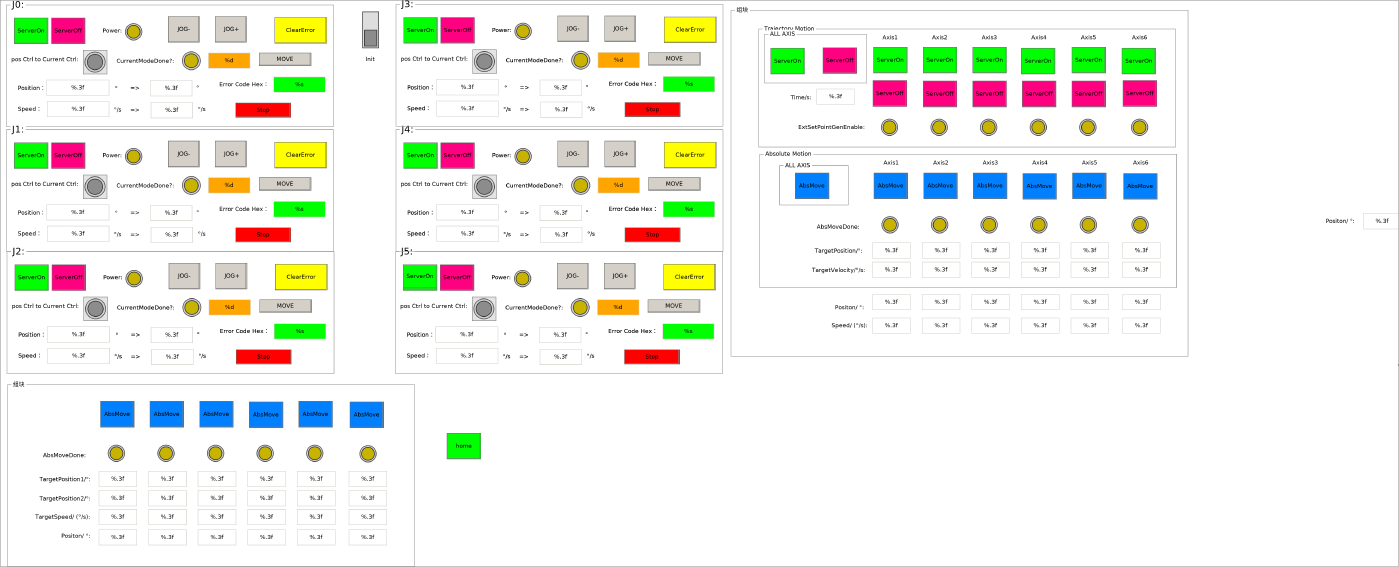
VISUALIZATION StatJoint_6Axis  // 2680x1087
    GroupBox (12,1 627x242), "J0:"
        Label (6,94 136x38), "pos Ctrl to Current Ctrl:"
        Label (13,192 64x32), "Speed："
        Label (224,191 45x38), "=>"
        Textfield (77,152 120x30), "%.3f", text variable: MAIN.AxisInfo[0].PositionCmd
        Label (198,154 22x29), "°"
        Textfield (78,193 119x30), "%.3f", text variable: MAIN.AxisMotionPara[0].TargetVelocity
            OnMouseClick: write the text variable via VisuDialogs.Numpad
        Label (193,195 37x29), "°/s"
        Button (86,33 65x50), "ServerOff", input disabled if: NOT MAIN.AxisOp[0].AxisInfo.AxisStatus.Ready
            toggle MAIN.HMI_AxisEnable[0]
        Button (514,32 100x50), "ClearError"
            tap MAIN.HMI_Axis_reset[0]
        Label (173,43 60x30), "Power:"
        Label (261,47 40x30)
        Button (310,30 60x50), "JOG-"
            tap MAIN.HMI_AxisJogBackwards[0]
        Button (400,30 60x50), "JOG+"
            tap MAIN.HMI_AxisJogFoward[0]
        Textfield (276,153 80x30), "%.3f", text variable: MAIN.AxisInfo[0].ActualPosition
        Label (354,153 22x29), "°"
        Label (354,194 37x29), "°/s"
        Textfield (277,195 80x30), "%.3f", text variable: MAIN.AxisInfo[0].ActualVelocity
        Textfield (387,100 80x30), "%d", text variable: MAIN.HMI_TargetTorque[0]
            OnMouseClick: write the text variable via VisuDialogs.Numpad
        Button (484,100 100x25), "MOVE"
            toggle MAIN.HMI_CurrentControlMove[0]
        Label (406,146 99x30), "Error Code Hex："
        Textfield (512,146 99x30), "%s", text variable: MAIN.AxisOp[0].AxisInfo.ErrId_Hex
        Label (224,149 45x38), "=>"
        Button (15,33 65x50), "ServerOn", input disabled if: NOT MAIN.AxisOp[0].AxisInfo.AxisStatus.Ready
            toggle MAIN.HMI_AxisEnable[0]
        PushSwitchLed (146,95 48x46), variable: MAIN.HMI_CurrentControlOfEnable[0], behaviour: TOGGLE, style: Switch-PushSwitchLed-Gray
        Label (18,149 62x38), "Position："
        Button (439,196 106x28), "Stop"
            tap MAIN.HMI_AxisStop[0]
        Lamp1 (225,40 38x40), variable: MAIN.AxisOp[0].AxisInfo.AxisStatus.Enabled, style: Lamp-Lamp1-Yellow
        Label (209,97 115x38), "CurrentModeDone?:"
        Lamp1 (334,94 41x43), variable: MAIN.HMI_AxisCurrentControlFlag[0], style: Lamp-Lamp1-Yellow
        Textfield (78,625 120x30), "%.3f", text variable: MAIN.AxisInfo[0].PositionCmd
        Label (199,627 22x29), "°"
        Label (14,665 64x32), "Speed："
        Textfield (79,666 119x30), "%.3f", text variable: MAIN.AxisMotionPara[0].TargetVelocity
            OnMouseClick: write the text variable via VisuDialogs.Numpad
        Label (194,668 37x29), "°/s"
        Button (87,506 65x50), "ServerOff", input disabled if: NOT MAIN.AxisOp[0].AxisInfo.AxisStatus.Ready
            toggle MAIN.HMI_AxisEnable[0]
        Button (515,505 100x50), "ClearError"
            tap MAIN.HMI_Axis_reset[0]
        Label (174,516 60x30), "Power:"
        Label (262,520 40x30)
        Button (311,503 60x50), "JOG-"
            tap MAIN.HMI_AxisJogBackwards[0]
        Button (401,503 60x50), "JOG+"
            tap MAIN.HMI_AxisJogFoward[0]
        Textfield (277,626 80x30), "%.3f", text variable: MAIN.AxisInfo[0].ActualPosition
        Label (355,626 22x29), "°"
        Label (355,667 37x29), "°/s"
        Textfield (278,668 80x30), "%.3f", text variable: MAIN.AxisInfo[0].ActualVelocity
        Textfield (388,573 80x30), "%d", text variable: MAIN.HMI_TargetTorque[0]
            OnMouseClick: write the text variable via VisuDialogs.Numpad
        Button (485,573 100x25), "MOVE"
            tap MAIN.HMI_CurrentControlMove[0]
        Label (407,619 99x30), "Error Code Hex："
        Textfield (513,619 99x30), "%s", text variable: MAIN.AxisOp[0].AxisInfo.ErrId_Hex
        Label (225,622 45x38), "=>"
        Label (225,664 45x38), "=>"
        Button (16,506 65x50), "ServerOn", input disabled if: NOT MAIN.AxisOp[0].AxisInfo.AxisStatus.Ready
            toggle MAIN.HMI_AxisEnable[0]
        PushSwitchLed (147,568 48x46), variable: MAIN.HMI_CurrentControlOfEnable[0], behaviour: TOGGLE, style: Switch-PushSwitchLed-Gray
        Label (19,622 62x38), "Position："
        Button (440,669 106x28), "Stop"
            tap MAIN.HMI_AxisStop[0]
        Lamp1 (226,513 38x40), variable: MAIN.AxisOp[0].AxisInfo.AxisStatus.Enabled, style: Lamp-Lamp1-Yellow
        Label (210,570 115x38), "CurrentModeDone?:"
        Lamp1 (335,567 41x43), variable: MAIN.HMI_AxisCurrentControlFlag[0], style: Lamp-Lamp1-Yellow
    DipSwitch (675,22 70x70), variable: MAIN.SiasunServoTestStart, behaviour: TOGGLE, style: Switch-DipSwitch-Gray
    Label (661,100 97x27), "Init"
    GroupBox (12,240 627x242), "J1:"
        Label (6,94 136x38), "pos Ctrl to Current Ctrl:"
        Textfield (77,152 120x30), "%.3f", text variable: MAIN.AxisInfo[1].PositionCmd
        Label (198,154 22x29), "°"
        Label (13,192 64x32), "Speed："
        Textfield (78,193 119x30), "%.3f", text variable: MAIN.AxisMotionPara[1].TargetVelocity
            OnMouseClick: write the text variable via VisuDialogs.Numpad
        Label (193,195 37x29), "°/s"
        Button (86,33 65x50), "ServerOff", input disabled if: NOT MAIN.AxisOp[1].AxisInfo.AxisStatus.Ready
            toggle MAIN.HMI_AxisEnable[1]
        Label (173,43 60x30), "Power:"
        Label (261,47 40x30)
        Button (310,30 60x50), "JOG-"
            tap MAIN.HMI_AxisJogBackwards[1]
        Button (400,30 60x50), "JOG+"
            tap MAIN.HMI_AxisJogFoward[1]
        Textfield (276,153 80x30), "%.3f", text variable: MAIN.AxisInfo[1].ActualPosition
        Label (354,153 22x29), "°"
        Label (354,194 37x29), "°/s"
        Textfield (277,195 80x30), "%.3f", text variable: MAIN.AxisInfo[1].ActualVelocity
        Textfield (387,100 80x30), "%d", text variable: MAIN.HMI_TargetTorque[1]
            OnMouseClick: write the text variable via VisuDialogs.Numpad
        Button (484,100 100x25), "MOVE"
            toggle MAIN.HMI_CurrentControlMove[1]
        Label (406,146 99x30), "Error Code Hex："
        Textfield (512,146 99x30), "%s", text variable: MAIN.AxisOp[1].AxisInfo.ErrId_Hex
        Label (224,149 45x38), "=>"
        Label (224,191 45x38), "=>"
        Button (15,33 65x50), "ServerOn", input disabled if: NOT MAIN.AxisOp[1].AxisInfo.AxisStatus.Ready
            toggle MAIN.HMI_AxisEnable[1]
        PushSwitchLed (146,95 48x46), variable: MAIN.HMI_CurrentControlOfEnable[1], behaviour: TOGGLE, style: Switch-PushSwitchLed-Gray
        Label (18,149 62x38), "Position："
        Button (439,196 106x28), "Stop"
            tap MAIN.HMI_AxisStop[1]
        Lamp1 (225,40 38x40), variable: MAIN.AxisOp[1].AxisInfo.AxisStatus.Enabled, style: Lamp-Lamp1-Yellow
        Label (209,97 115x38), "CurrentModeDone?:"
        Lamp1 (334,94 41x43), variable: MAIN.HMI_AxisCurrentControlFlag[1], style: Lamp-Lamp1-Yellow
        Button (514,32 100x50), "ClearError"
            tap MAIN.HMI_Axis_reset[1]
    GroupBox (13,474 627x242), "J2:"
        Label (6,94 136x38), "pos Ctrl to Current Ctrl:"
        Textfield (77,152 120x30), "%.3f", text variable: MAIN.AxisInfo[2].PositionCmd
        Label (198,154 22x29), "°"
        Label (13,192 64x32), "Speed："
        Textfield (78,193 119x30), "%.3f", text variable: MAIN.AxisMotionPara[2].TargetVelocity
            OnMouseClick: write the text variable via VisuDialogs.Numpad
        Label (193,195 37x29), "°/s"
        Button (86,33 65x50), "ServerOff", input disabled if: NOT MAIN.AxisOp[2].AxisInfo.AxisStatus.Ready
            toggle MAIN.HMI_AxisEnable[2]
        Button (514,32 100x50), "ClearError"
            tap MAIN.HMI_Axis_reset[2]
        Label (173,43 60x30), "Power:"
        Label (261,47 40x30)
        Button (310,30 60x50), "JOG-"
            tap MAIN.HMI_AxisJogBackwards[2]
        Button (400,30 60x50), "JOG+"
            tap MAIN.HMI_AxisJogFoward[2]
        Textfield (276,153 80x30), "%.3f", text variable: MAIN.AxisInfo[2].ActualPosition
        Label (354,153 22x29), "°"
        Label (354,194 37x29), "°/s"
        Textfield (277,195 80x30), "%.3f", text variable: MAIN.AxisInfo[2].ActualVelocity
        Textfield (387,100 80x30), "%d", text variable: MAIN.HMI_TargetTorque[2]
            OnMouseClick: write the text variable via VisuDialogs.Numpad
        Button (484,100 100x25), "MOVE"
            toggle MAIN.HMI_CurrentControlMove[2]
        Label (406,146 99x30), "Error Code Hex："
        Textfield (512,146 99x30), "%s", text variable: MAIN.AxisOp[2].AxisInfo.ErrId_Hex
        Label (224,149 45x38), "=>"
        Label (224,191 45x38), "=>"
        Button (15,33 65x50), "ServerOn", input disabled if: NOT MAIN.AxisOp[2].AxisInfo.AxisStatus.Ready
            toggle MAIN.HMI_AxisEnable[2]
        PushSwitchLed (146,95 48x46), variable: MAIN.HMI_CurrentControlOfEnable[2], behaviour: TOGGLE, style: Switch-PushSwitchLed-Gray
        Label (18,149 62x38), "Position："
        Button (439,196 106x28), "Stop"
            tap MAIN.HMI_AxisStop[2]
        Lamp1 (225,40 38x40), variable: MAIN.AxisOp[2].AxisInfo.AxisStatus.Enabled, style: Lamp-Lamp1-Yellow
        Label (209,97 115x38), "CurrentModeDone?:"
        Lamp1 (334,94 41x43), variable: MAIN.HMI_AxisCurrentControlFlag[2], style: Lamp-Lamp1-Yellow
        Textfield (821,152 120x30), "%.3f", text variable: MAIN.AxisInfo[0].PositionCmd
        Label (942,154 22x29), "°"
        Label (757,192 64x32), "Speed："
        Textfield (822,193 119x30), "%.3f", text variable: MAIN.AxisMotionPara[0].TargetVelocity
            OnMouseClick: write the text variable via VisuDialogs.Numpad
        Label (937,195 37x29), "°/s"
        Button (830,33 65x50), "ServerOff", input disabled if: NOT MAIN.AxisOp[0].AxisInfo.AxisStatus.Ready
            toggle MAIN.HMI_AxisEnable[0]
        Button (1258,32 100x50), "ClearError"
            tap MAIN.HMI_Axis_reset[0]
        Label (917,43 60x30), "Power:"
        Label (1005,47 40x30)
        Button (1054,30 60x50), "JOG-"
            tap MAIN.HMI_AxisJogBackwards[0]
        Button (1144,30 60x50), "JOG+"
            tap MAIN.HMI_AxisJogFoward[0]
        Textfield (1020,153 80x30), "%.3f", text variable: MAIN.AxisInfo[0].ActualPosition
        Label (1098,153 22x29), "°"
        Label (1098,194 37x29), "°/s"
        Textfield (1021,195 80x30), "%.3f", text variable: MAIN.AxisInfo[0].ActualVelocity
        Textfield (1131,100 80x30), "%d", text variable: MAIN.HMI_TargetTorque[0]
            OnMouseClick: write the text variable via VisuDialogs.Numpad
        Button (1228,100 100x25), "MOVE"
            tap MAIN.HMI_CurrentControlMove[0]
        Label (1150,146 99x30), "Error Code Hex："
        Textfield (1256,146 99x30), "%s", text variable: MAIN.AxisOp[0].AxisInfo.ErrId_Hex
        Label (968,149 45x38), "=>"
        Label (968,191 45x38), "=>"
        Button (759,33 65x50), "ServerOn", input disabled if: NOT MAIN.AxisOp[0].AxisInfo.AxisStatus.Ready
            toggle MAIN.HMI_AxisEnable[0]
        PushSwitchLed (890,95 48x46), variable: MAIN.HMI_CurrentControlOfEnable[0], behaviour: TOGGLE, style: Switch-PushSwitchLed-Gray
        Label (762,149 62x38), "Position："
        Button (1183,196 106x28), "Stop"
            tap MAIN.HMI_AxisStop[0]
        Lamp1 (969,40 38x40), variable: MAIN.AxisOp[0].AxisInfo.AxisStatus.Enabled, style: Lamp-Lamp1-Yellow
        Label (953,97 115x38), "CurrentModeDone?:"
        Lamp1 (1078,94 41x43), variable: MAIN.HMI_AxisCurrentControlFlag[0], style: Lamp-Lamp1-Yellow
    GroupBox (757,474 627x242), "J5:"
        Label (6,94 136x38), "pos Ctrl to Current Ctrl:"
        Textfield (77,152 120x30), "%.3f", text variable: MAIN.AxisInfo[5].PositionCmd
        Label (198,154 22x29), "°"
        Label (13,192 64x32), "Speed："
        Textfield (78,193 119x30), "%.3f", text variable: MAIN.AxisMotionPara[5].TargetVelocity
            OnMouseClick: write the text variable via VisuDialogs.Numpad
        Label (193,195 37x29), "°/s"
        Button (86,33 65x50), "ServerOff", input disabled if: NOT MAIN.AxisOp[5].AxisInfo.AxisStatus.Ready
            toggle MAIN.HMI_AxisEnable[5]
        Button (514,32 100x50), "ClearError"
            tap MAIN.HMI_Axis_reset[5]
        Label (173,43 60x30), "Power:"
        Label (261,47 40x30)
        Button (310,30 60x50), "JOG-"
            tap MAIN.HMI_AxisJogBackwards[5]
        Button (400,30 60x50), "JOG+"
            tap MAIN.HMI_AxisJogFoward[5]
        Textfield (276,153 80x30), "%.3f", text variable: MAIN.AxisInfo[5].ActualPosition
        Label (354,153 22x29), "°"
        Label (354,194 37x29), "°/s"
        Textfield (277,195 80x30), "%.3f", text variable: MAIN.AxisInfo[5].ActualVelocity
        Textfield (387,100 80x30), "%d", text variable: MAIN.HMI_TargetTorque[5]
            OnMouseClick: write the text variable via VisuDialogs.Numpad
        Button (484,100 100x25), "MOVE"
            toggle MAIN.HMI_CurrentControlMove[5]
        Label (406,146 99x30), "Error Code Hex："
        Textfield (512,146 99x30), "%s", text variable: MAIN.AxisOp[5].AxisInfo.ErrId_Hex
        Label (224,149 45x38), "=>"
        Label (224,191 45x38), "=>"
        Button (15,33 65x45), "ServerOn", input disabled if: NOT MAIN.AxisOp[5].AxisInfo.AxisStatus.Ready
            toggle MAIN.HMI_AxisEnable[5]
        PushSwitchLed (146,95 48x46), variable: MAIN.HMI_CurrentControlOfEnable[5], behaviour: TOGGLE, style: Switch-PushSwitchLed-Gray
        Label (18,149 62x38), "Position："
        Button (439,196 106x28), "Stop"
            tap MAIN.HMI_AxisStop[5]
        Lamp1 (225,40 38x40), variable: MAIN.AxisOp[5].AxisInfo.AxisStatus.Enabled, style: Lamp-Lamp1-Yellow
        Label (209,97 115x38), "CurrentModeDone?:"
        Lamp1 (334,94 41x43), variable: MAIN.HMI_AxisCurrentControlFlag[5], style: Lamp-Lamp1-Yellow
        Textfield (78,-82 120x30), "%.3f", text variable: MAIN.AxisInfo[0].PositionCmd
        Label (199,-80 22x29), "°"
        Label (14,-42 64x32), "Speed："
        Textfield (79,-41 119x30), "%.3f", text variable: MAIN.AxisMotionPara[0].TargetVelocity
            OnMouseClick: write the text variable via VisuDialogs.Numpad
        Label (194,-39 37x29), "°/s"
        Button (87,-201 65x50), "ServerOff", input disabled if: NOT MAIN.AxisOp[0].AxisInfo.AxisStatus.Ready
            toggle MAIN.HMI_AxisEnable[0]
        Button (515,-202 100x50), "ClearError"
            tap MAIN.HMI_Axis_reset[0]
        Label (174,-191 60x30), "Power:"
        Label (262,-187 40x30)
        Button (311,-204 60x50), "JOG-"
            tap MAIN.HMI_AxisJogBackwards[0]
        Button (401,-204 60x50), "JOG+"
            tap MAIN.HMI_AxisJogFoward[0]
        Textfield (277,-81 80x30), "%.3f", text variable: MAIN.AxisInfo[0].ActualPosition
        Label (355,-81 22x29), "°"
        Label (355,-40 37x29), "°/s"
        Textfield (278,-39 80x30), "%.3f", text variable: MAIN.AxisInfo[0].ActualVelocity
        Textfield (388,-134 80x30), "%d", text variable: MAIN.HMI_TargetTorque[0]
            OnMouseClick: write the text variable via VisuDialogs.Numpad
        Button (485,-134 100x25), "MOVE"
            tap MAIN.HMI_CurrentControlMove[0]
        Label (407,-88 99x30), "Error Code Hex："
        Textfield (513,-88 99x30), "%s", text variable: MAIN.AxisOp[0].AxisInfo.ErrId_Hex
        Label (225,-85 45x38), "=>"
        Label (225,-43 45x38), "=>"
        Button (16,-201 65x50), "ServerOn", input disabled if: NOT MAIN.AxisOp[0].AxisInfo.AxisStatus.Ready
            toggle MAIN.HMI_AxisEnable[0]
        PushSwitchLed (147,-139 48x46), variable: MAIN.HMI_CurrentControlOfEnable[0], behaviour: TOGGLE, style: Switch-PushSwitchLed-Gray
        Label (19,-85 62x38), "Position："
        Button (440,-38 106x28), "Stop"
            tap MAIN.HMI_AxisStop[0]
        Lamp1 (226,-194 38x40), variable: MAIN.AxisOp[0].AxisInfo.AxisStatus.Enabled, style: Lamp-Lamp1-Yellow
        Label (210,-137 115x38), "CurrentModeDone?:"
        Lamp1 (335,-140 41x43), variable: MAIN.HMI_AxisCurrentControlFlag[0], style: Lamp-Lamp1-Yellow
    GroupBox (758,240 627x242), "J4:"
        Label (6,94 136x38), "pos Ctrl to Current Ctrl:"
        Textfield (77,152 120x30), "%.3f", text variable: MAIN.AxisInfo[4].PositionCmd
        Label (198,154 22x29), "°"
        Label (13,192 64x32), "Speed："
        Textfield (78,193 119x30), "%.3f", text variable: MAIN.AxisMotionPara[4].TargetVelocity
            OnMouseClick: write the text variable via VisuDialogs.Numpad
        Label (193,195 37x29), "°/s"
        Button (86,33 65x50), "ServerOff", input disabled if: NOT MAIN.AxisOp[4].AxisInfo.AxisStatus.Ready
            toggle MAIN.HMI_AxisEnable[4]
        Button (514,32 100x50), "ClearError"
            tap MAIN.HMI_Axis_reset[4]
        Label (173,43 60x30), "Power:"
        Label (261,47 40x30)
        Button (310,30 60x50), "JOG-"
            tap MAIN.HMI_AxisJogBackwards[4]
        Button (400,30 60x50), "JOG+"
            tap MAIN.HMI_AxisJogFoward[4]
        Textfield (276,153 80x30), "%.3f", text variable: MAIN.AxisInfo[4].ActualPosition
        Label (354,153 22x29), "°"
        Label (354,194 37x29), "°/s"
        Textfield (277,195 80x30), "%.3f", text variable: MAIN.AxisInfo[4].ActualVelocity
        Textfield (387,100 80x30), "%d", text variable: MAIN.HMI_TargetTorque[4]
            OnMouseClick: write the text variable via VisuDialogs.Numpad
        Button (484,100 100x25), "MOVE"
            toggle MAIN.HMI_CurrentControlMove[4]
        Label (406,146 99x30), "Error Code Hex："
        Textfield (512,146 99x30), "%s", text variable: MAIN.AxisOp[4].AxisInfo.ErrId_Hex
        Label (224,149 45x38), "=>"
        Label (224,191 45x38), "=>"
        Button (15,33 65x50), "ServerOn", input disabled if: NOT MAIN.AxisOp[4].AxisInfo.AxisStatus.Ready
            toggle MAIN.HMI_AxisEnable[4]
        PushSwitchLed (146,95 48x46), variable: MAIN.HMI_CurrentControlOfEnable[4], behaviour: TOGGLE, style: Switch-PushSwitchLed-Gray
        Label (18,149 62x38), "Position："
        Button (439,196 106x28), "Stop"
            tap MAIN.HMI_AxisStop[4]
        Lamp1 (225,40 38x40), variable: MAIN.AxisOp[4].AxisInfo.AxisStatus.Enabled, style: Lamp-Lamp1-Yellow
        Label (209,97 115x38), "CurrentModeDone?:"
        Lamp1 (334,94 41x43), variable: MAIN.HMI_AxisCurrentControlFlag[4], style: Lamp-Lamp1-Yellow
        Group (13,-210 601x199)
            Textfield (64,122 120x30), "%.3f", text variable: MAIN.AxisInfo[0].PositionCmd
            Label (185,124 22x29), "°"
            Label (0,162 64x32), "Speed："
            Textfield (65,163 119x30), "%.3f", text variable: MAIN.AxisMotionPara[0].TargetVelocity
                OnMouseClick: write the text variable via VisuDialogs.Numpad
            Label (180,165 37x29), "°/s"
            Button (73,3 65x50), "ServerOff", input disabled if: NOT MAIN.AxisOp[0].AxisInfo.AxisStatus.Ready
                toggle MAIN.HMI_AxisEnable[0]
            Button (501,2 100x50), "ClearError"
                tap MAIN.HMI_Axis_reset[0]
            Label (160,13 60x30), "Power:"
            Label (248,17 40x30)
            Button (297,0 60x50), "JOG-"
                tap MAIN.HMI_AxisJogBackwards[0]
            Button (387,0 60x50), "JOG+"
                tap MAIN.HMI_AxisJogFoward[0]
            Textfield (263,123 80x30), "%.3f", text variable: MAIN.AxisInfo[0].ActualPosition
            Label (341,123 22x29), "°"
            Label (341,164 37x29), "°/s"
            Textfield (264,165 80x30), "%.3f", text variable: MAIN.AxisInfo[0].ActualVelocity
            Textfield (374,70 80x30), "%d", text variable: MAIN.HMI_TargetTorque[0]
                OnMouseClick: write the text variable via VisuDialogs.Numpad
            Button (471,70 100x25), "MOVE"
                tap MAIN.HMI_CurrentControlMove[0]
            Label (393,116 99x30), "Error Code Hex："
            Textfield (499,116 99x30), "%s", text variable: MAIN.AxisOp[0].AxisInfo.ErrId_Hex
            Label (211,119 45x38), "=>"
            Label (211,161 45x38), "=>"
            Button (2,3 65x50), "ServerOn", input disabled if: NOT MAIN.AxisOp[0].AxisInfo.AxisStatus.Ready
                toggle MAIN.HMI_AxisEnable[0]
            PushSwitchLed (133,65 48x46), variable: MAIN.HMI_CurrentControlOfEnable[0], behaviour: TOGGLE, style: Switch-PushSwitchLed-Gray
            Label (5,119 62x38), "Position："
            Button (426,166 106x28), "Stop"
                tap MAIN.HMI_AxisStop[0]
            Lamp1 (212,10 38x40), variable: MAIN.AxisOp[0].AxisInfo.AxisStatus.Enabled, style: Lamp-Lamp1-Yellow
            Label (196,67 115x38), "CurrentModeDone?:"
            Lamp1 (321,64 41x43), variable: MAIN.HMI_AxisCurrentControlFlag[0], style: Lamp-Lamp1-Yellow
    GroupBox (758,0 627x242), "J3:"
        Label (6,94 136x38), "pos Ctrl to Current Ctrl:"
        Textfield (77,152 120x30), "%.3f", text variable: MAIN.AxisInfo[3].PositionCmd
        Label (198,154 22x29), "°"
        Label (13,192 64x32), "Speed："
        Textfield (78,193 119x30), "%.3f", text variable: MAIN.AxisMotionPara[3].TargetVelocity
            OnMouseClick: write the text variable via VisuDialogs.Numpad
        Label (193,195 37x29), "°/s"
        Button (86,33 65x50), "ServerOff", input disabled if: NOT MAIN.AxisOp[3].AxisInfo.AxisStatus.Ready
            toggle MAIN.HMI_AxisEnable[3]
        Button (514,32 100x50), "ClearError"
            tap MAIN.HMI_Axis_reset[3]
        Label (173,43 60x30), "Power:"
        Label (261,47 40x30)
        Button (310,30 60x50), "JOG-"
            tap MAIN.HMI_AxisJogBackwards[3]
        Button (400,30 60x50), "JOG+"
            tap MAIN.HMI_AxisJogFoward[3]
        Textfield (276,153 80x30), "%.3f", text variable: MAIN.AxisInfo[3].ActualPosition
        Label (354,153 22x29), "°"
        Label (354,194 37x29), "°/s"
        Textfield (277,195 80x30), "%.3f", text variable: MAIN.AxisInfo[3].ActualVelocity
        Textfield (387,100 80x30), "%d", text variable: MAIN.HMI_TargetTorque[3]
            OnMouseClick: write the text variable via VisuDialogs.Numpad
        Button (484,100 100x25), "MOVE"
            toggle MAIN.HMI_CurrentControlMove[3]
        Label (406,146 99x30), "Error Code Hex："
        Textfield (512,146 99x30), "%s", text variable: MAIN.AxisOp[3].AxisInfo.ErrId_Hex
        Label (224,149 45x38), "=>"
        Label (224,191 45x38), "=>"
        Button (15,33 65x50), "ServerOn", input disabled if: NOT MAIN.AxisOp[3].AxisInfo.AxisStatus.Ready
            toggle MAIN.HMI_AxisEnable[3]
        PushSwitchLed (146,95 48x46), variable: MAIN.HMI_CurrentControlOfEnable[3], behaviour: TOGGLE, style: Switch-PushSwitchLed-Gray
        Label (18,149 62x38), "Position："
        Button (439,196 106x28), "Stop"
            tap MAIN.HMI_AxisStop[3]
        Lamp1 (225,40 38x40), variable: MAIN.AxisOp[3].AxisInfo.AxisStatus.Enabled, style: Lamp-Lamp1-Yellow
        Label (209,97 115x38), "CurrentModeDone?:"
        Lamp1 (334,94 41x43), variable: MAIN.HMI_AxisCurrentControlFlag[3], style: Lamp-Lamp1-Yellow
    Button (2678,700 2x0)
    GroupBox (1400,11 876x672), "组块"
        GroupBox (53,36 799x235), "Trajectory Motion"
            Button (220,43 65x50), "ServerOn"
                OnMouseClick: execute { Main.HMI_Tra_Motion[0]:=TRUE; }
            Button (219,107 65x50), "ServerOff"
                OnMouseClick: execute { Main.HMI_Tra_Motion[0]:=FALSE; }
            Lamp1 (232,177 38x40), variable: MAIN.AxisOp[0].AxisDrive.AxisExtSetPointGenEnable.Enabled, style: Lamp-Lamp1-Yellow
            Lamp1 (327,177 38x40), variable: MAIN.AxisOp[1].AxisDrive.AxisExtSetPointGenEnable.Enabled, style: Lamp-Lamp1-Yellow
            Lamp1 (422,177 38x40), variable: MAIN.AxisOp[2].AxisDrive.AxisExtSetPointGenEnable.Enabled, style: Lamp-Lamp1-Yellow
            Lamp1 (517,177 38x40), variable: MAIN.AxisOp[3].AxisDrive.AxisExtSetPointGenEnable.Enabled, style: Lamp-Lamp1-Yellow
            Lamp1 (612,177 38x40), variable: MAIN.AxisOp[4].AxisDrive.AxisExtSetPointGenEnable.Enabled, style: Lamp-Lamp1-Yellow
            Lamp1 (711,177 38x40), variable: MAIN.AxisOp[5].AxisDrive.AxisExtSetPointGenEnable.Enabled, style: Lamp-Lamp1-Yellow
            Button (315,43 65x50), "ServerOn"
                OnMouseClick: execute { Main.HMI_Tra_Motion[1]:=TRUE; }
            Button (410,43 65x50), "ServerOn"
                OnMouseClick: execute { Main.HMI_Tra_Motion[2]:=TRUE; }
            Button (600,43 65x50), "ServerOn"
                OnMouseClick: execute { Main.HMI_Tra_Motion[4]:=TRUE; }
            GroupBox (11,10 196x102), "ALL AXIS"
                Button (112,34 65x50), "ServerOff"
                    OnMouseClick: execute {
                        Main.HMI_Tra_Motion[0]:=FALSE;
                        Main.HMI_Tra_Motion[1]:=FALSE;
                        Main.HMI_Tra_Motion[2]:=FALSE;
                        Main.HMI_Tra_Motion[3]:=FALSE;
                        Main.HMI_Tra_Motion[4]:=FALSE;
                        Main.HMI_Tra_Motion[5]:=FALSE;
                    }
                Button (12,35 65x50), "ServerOn"
                    OnMouseClick: execute {
                        Main.HMI_Tra_Motion[0]:=TRUE;
                        Main.HMI_Tra_Motion[1]:=TRUE;
                        Main.HMI_Tra_Motion[2]:=TRUE;
                        Main.HMI_Tra_Motion[3]:=TRUE;
                        Main.HMI_Tra_Motion[4]:=TRUE;
                        Main.HMI_Tra_Motion[5]:=TRUE;
                    }
            Label (229,10 47x30), "Axis1"
            Label (324,10 47x30), "Axis2"
            Label (419,10 47x30), "Axis3"
            Label (514,10 47x30), "Axis4"
            Label (609,10 47x30), "Axis5"
            Label (707,10 47x30), "Axis6"
            Textfield (111,123 73x30), "%.3f", text variable: MAIN.AxisOp[0].AxisDrive.timer
            Label (58,125 47x30), "Time/s:"
            Label (72,182 136x30), "ExtSetPointGenEnable:"
            Button (315,108 65x50), "ServerOff"
                OnMouseClick: execute { Main.HMI_Tra_Motion[1]:=FALSE; }
            Button (410,108 65x50), "ServerOff"
                OnMouseClick: execute { Main.HMI_Tra_Motion[2]:=FALSE; }
            Button (505,108 65x50), "ServerOff"
                OnMouseClick: execute { Main.HMI_Tra_Motion[3]:=FALSE; }
            Button (600,108 65x50), "ServerOff"
                OnMouseClick: execute { Main.HMI_Tra_Motion[4]:=FALSE; }
            Button (698,107 65x50), "ServerOff"
                OnMouseClick: execute { Main.HMI_Tra_Motion[5]:=FALSE; }
            Button (503,45 65x50), "ServerOn"
                OnMouseClick: execute {  }
                OnMouseClick: execute { Main.HMI_Tra_Motion[3]:=TRUE; }
            Button (696,45 65x50), "ServerOn"
                OnMouseClick: execute { Main.HMI_Tra_Motion[5]:=TRUE; }
        GroupBox (55,276 799x264), "Absolute Motion"
            Label (229,10 47x30), "Axis1"
            Label (324,10 47x30), "Axis2"
            Label (419,10 47x30), "Axis3"
            Label (514,10 47x30), "Axis4"
            Label (609,10 47x30), "Axis5"
            Label (707,10 47x30), "Axis6"
            Textfield (1156,122 73x30), "%.3f", text variable: MAIN.AxisOP[0].AxisRef.NcToPlc.ActPos
            Textfield (1346,122 73x30), "%.3f", text variable: MAIN.AxisOP[2].AxisRef.NcToPlc.ActPos
            Textfield (1251,122 73x30), "%.3f", text variable: MAIN.AxisOP[1].AxisRef.NcToPlc.ActPos
            Textfield (1441,122 73x30), "%.3f", text variable: MAIN.AxisOP[3].AxisRef.NcToPlc.ActPos
            Textfield (1536,122 73x30), "%.3f", text variable: MAIN.AxisOP[4].AxisRef.NcToPlc.ActPos
            Textfield (1635,122 73x30), "%.3f", text variable: MAIN.AxisOP[5].AxisRef.NcToPlc.ActPos
            Label (1076,122 73x30), "Positon/ °:"
            GroupBox (38,22 132x84), "ALL AXIS"
                Button (30,22 65x50), "AbsMove"
                    OnMouseClick: execute {
                        Main.HMI_Abs_Motion[0]:=TRUE;
                        Main.HMI_Abs_Motion[1]:=TRUE;
                        Main.HMI_Abs_Motion[2]:=TRUE;
                        Main.HMI_Abs_Motion[3]:=TRUE;
                        Main.HMI_Abs_Motion[4]:=TRUE;
                        Main.HMI_Abs_Motion[5]:=TRUE;
                    }
            Button (219,44 65x50), "AbsMove"
                OnMouseClick: execute { main.HMI_Abs_Motion[0]:=TRUE; }
            Lamp1 (231,124 38x40), variable: MAIN.AxisOP[0].AxisDrive.MoveAbsolute.Active, style: Lamp-Lamp1-Yellow
            Lamp1 (326,124 38x40), variable: MAIN.AxisOP[1].AxisDrive.MoveAbsolute.Active, style: Lamp-Lamp1-Yellow
            Lamp1 (421,124 38x40), variable: MAIN.AxisOP[2].AxisDrive.MoveAbsolute.Active, style: Lamp-Lamp1-Yellow
            Lamp1 (516,124 38x40), variable: MAIN.AxisOP[3].AxisDrive.MoveAbsolute.Active, style: Lamp-Lamp1-Yellow
            Lamp1 (611,124 38x40), variable: MAIN.AxisOP[4].AxisDrive.MoveAbsolute.Active, style: Lamp-Lamp1-Yellow
            Lamp1 (710,124 38x40), variable: MAIN.AxisOP[5].AxisDrive.MoveAbsolute.Active, style: Lamp-Lamp1-Yellow
            Button (314,44 65x50), "AbsMove"
                OnMouseClick: execute { Main.HMI_Abs_Motion[1]:=TRUE; }
            Button (409,44 65x50), "AbsMove"
                OnMouseClick: execute { Main.HMI_Abs_Motion[2]:=TRUE; }
            Button (599,44 65x50), "AbsMove"
                OnMouseClick: execute { Main.HMI_Abs_Motion[4]:=TRUE; }
            Label (94,133 113x30), "AbsMoveDone:"
            Button (504,45 65x50), "AbsMove"
                OnMouseClick: execute {  }
                OnMouseClick: execute { Main.HMI_Abs_Motion[3]:=TRUE; }
            Button (697,45 65x50), "AbsMove"
                OnMouseClick: execute { Main.HMI_Abs_Motion[5]:=TRUE; }
            Textfield (216,178 73x30), "%.3f", text variable: MAIN.AxisOP[0].AxisMotionPara.TargetPosition
                OnMouseClick: write the text variable via VisuDialogs.Numpad
            Textfield (406,178 73x30), "%.3f", text variable: MAIN.AxisOP[2].AxisMotionPara.TargetPosition
                OnMouseClick: write the text variable via VisuDialogs.Numpad
            Textfield (311,178 73x30), "%.3f", text variable: MAIN.AxisOP[1].AxisMotionPara.TargetPosition
                OnMouseClick: write the text variable via VisuDialogs.Numpad
            Textfield (501,178 73x30), "%.3f", text variable: MAIN.AxisOP[3].AxisMotionPara.TargetPosition
                OnMouseClick: write the text variable via VisuDialogs.Numpad
            Textfield (596,178 73x30), "%.3f", text variable: MAIN.AxisOP[4].AxisMotionPara.TargetPosition
                OnMouseClick: write the text variable via VisuDialogs.Numpad
            Textfield (695,178 73x30), "%.3f", text variable: MAIN.AxisOP[5].AxisMotionPara.TargetPosition
                OnMouseClick: write the text variable via VisuDialogs.Numpad
            Label (95,179 113x30), "TargetPosition/°:"
            Textfield (216,215 73x30), "%.3f", text variable: MAIN.AxisOP[0].AxisMotionPara.AbsMotion_Velocity
                OnMouseClick: write the text variable via VisuDialogs.Numpad
        Textfield (271,553 73x30), "%.3f", text variable: MAIN.AxisOP[0].AxisRef.NcToPlc.ActPos
        Textfield (461,553 73x30), "%.3f", text variable: MAIN.AxisOP[2].AxisRef.NcToPlc.ActPos
        Textfield (366,553 73x30), "%.3f", text variable: MAIN.AxisOP[1].AxisRef.NcToPlc.ActPos
        Textfield (556,553 73x30), "%.3f", text variable: MAIN.AxisOP[3].AxisRef.NcToPlc.ActPos
        Textfield (651,553 73x30), "%.3f", text variable: MAIN.AxisOP[4].AxisRef.NcToPlc.ActPos
        Textfield (750,553 73x30), "%.3f", text variable: MAIN.AxisOP[5].AxisRef.NcToPlc.ActPos
        Textfield (271,598 73x30), "%.3f", text variable: MAIN.AxisOP[0].AxisRef.NcToPlc.ActVelo
        Label (191,553 73x51), "Positon/ °:"
        Label (191,598 73x30), "Speed/ (°/s):"
        Textfield (461,598 73x30), "%.3f", text variable: MAIN.AxisOP[2].AxisRef.NcToPlc.ActVelo
        Textfield (366,598 73x30), "%.3f", text variable: MAIN.AxisOP[1].AxisRef.NcToPlc.ActVelo
        Textfield (556,598 73x30), "%.3f", text variable: MAIN.AxisOP[3].AxisRef.NcToPlc.ActVelo
        Textfield (651,598 73x30), "%.3f", text variable: MAIN.AxisOP[4].AxisRef.NcToPlc.ActVelo
        Textfield (750,598 73x30), "%.3f", text variable: MAIN.AxisOP[5].AxisRef.NcToPlc.ActVelo
    Textfield (1861,502 73x30), "%.3f", text variable: MAIN.AxisOP[2].AxisMotionPara.AbsMotion_Velocity
        OnMouseClick: write the text variable via VisuDialogs.Numpad
    Textfield (1766,502 73x30), "%.3f", text variable: MAIN.AxisOP[1].AxisMotionPara.AbsMotion_Velocity
        OnMouseClick: write the text variable via VisuDialogs.Numpad
    Textfield (1956,502 73x30), "%.3f", text variable: MAIN.AxisOP[3].AxisMotionPara.AbsMotion_Velocity
        OnMouseClick: write the text variable via VisuDialogs.Numpad
    Textfield (2051,502 73x30), "%.3f", text variable: MAIN.AxisOP[4].AxisMotionPara.AbsMotion_Velocity
        OnMouseClick: write the text variable via VisuDialogs.Numpad
    Textfield (2150,502 73x30), "%.3f", text variable: MAIN.AxisOP[5].AxisMotionPara.AbsMotion_Velocity
        OnMouseClick: write the text variable via VisuDialogs.Numpad
    Label (1550,503 113x30), "TargetVelocity/°/s:"
    GroupBox (14,729 780x358), "组块"
        Button (178,40 65x50), "AbsMove"
            OnMouseClick: execute { main.HMI_Reverse_Motion[0]:=TRUE; }
        Lamp1 (190,120 38x40), variable: MAIN.AxisOP[0].move_reverse_lamp, style: Lamp-Lamp1-Yellow
        Lamp1 (285,120 38x40), variable: MAIN.AxisOP[1].move_reverse_lamp, style: Lamp-Lamp1-Yellow
        Lamp1 (380,120 38x40), variable: MAIN.AxisOP[2].move_reverse_lamp, style: Lamp-Lamp1-Yellow
        Lamp1 (475,120 38x40), variable: MAIN.AxisOP[3].move_reverse_lamp, style: Lamp-Lamp1-Yellow
        Button (273,40 65x50), "AbsMove"
            OnMouseClick: execute { main.HMI_Reverse_Motion[1]:=TRUE; }
        Button (368,40 65x50), "AbsMove"
            OnMouseClick: execute { Main.HMI_Reverse_Motion[2]:=TRUE; }
        Button (558,40 65x50), "AbsMove"
            OnMouseClick: execute { Main.HMI_Reverse_Motion[4]:=TRUE; }
        Label (53,129 113x30), "AbsMoveDone:"
        Button (463,41 65x50), "AbsMove"
            OnMouseClick: execute { Main.HMI_Reverse_Motion[3]:=TRUE; }
        Button (656,41 65x50), "AbsMove"
            OnMouseClick: execute { Main.HMI_Reverse_Motion[5]:=TRUE; }
        Textfield (175,174 73x30), "%.3f", text variable: MAIN.AxisOP[0].AxisMotionPara.TargetPosition1
            OnMouseClick: write the text variable via VisuDialogs.Numpad
        Textfield (365,174 73x30), "%.3f", text variable: MAIN.AxisOP[2].AxisMotionPara.TargetPosition1
            OnMouseClick: write the text variable via VisuDialogs.Numpad
        Textfield (270,174 73x30), "%.3f", text variable: MAIN.AxisOP[1].AxisMotionPara.TargetPosition1
            OnMouseClick: write the text variable via VisuDialogs.Numpad
        Textfield (460,174 73x30), "%.3f", text variable: MAIN.AxisOP[3].AxisMotionPara.TargetPosition1
            OnMouseClick: write the text variable via VisuDialogs.Numpad
        Textfield (555,174 73x30), "%.3f", text variable: MAIN.AxisOP[4].AxisMotionPara.TargetPosition1
            OnMouseClick: write the text variable via VisuDialogs.Numpad
        Textfield (654,174 73x30), "%.3f", text variable: MAIN.AxisOP[5].AxisMotionPara.TargetPosition1
            OnMouseClick: write the text variable via VisuDialogs.Numpad
        Label (54,175 113x30), "TargetPosition1/°:"
        Textfield (175,211 73x30), "%.3f", text variable: MAIN.AxisOP[0].AxisMotionPara.TargetPosition2
            OnMouseClick: write the text variable via VisuDialogs.Numpad
        Textfield (175,286 73x30), "%.3f", text variable: MAIN.AxisOP[0].AxisRef.NcToPlc.ActPos
        Textfield (365,286 73x30), "%.3f", text variable: MAIN.AxisOP[2].AxisRef.NcToPlc.ActPos
        Textfield (270,286 73x30), "%.3f", text variable: MAIN.AxisOP[1].AxisRef.NcToPlc.ActPos
        Textfield (460,286 73x30), "%.3f", text variable: MAIN.AxisOP[3].AxisRef.NcToPlc.ActPos
        Textfield (555,286 73x30), "%.3f", text variable: MAIN.AxisOP[4].AxisRef.NcToPlc.ActPos
        Textfield (654,286 73x30), "%.3f", text variable: MAIN.AxisOP[5].AxisRef.NcToPlc.ActPos
        Textfield (175,247 73x30), "%.3f", text variable: MAIN.AxisOP[0].AxisMotionPara.ReverseMotion_Velocity
            OnMouseClick: write the text variable via VisuDialogs.Numpad
        Label (95,273 73x51), "Positon/ °:"
        Label (44,247 124x30), "TargetSpeed/ (°/s):"
        Textfield (365,247 73x30), "%.3f", text variable: MAIN.AxisOP[2].AxisMotionPara.ReverseMotion_Velocity
            OnMouseClick: write the text variable via VisuDialogs.Numpad
        Textfield (270,247 73x30), "%.3f", text variable: MAIN.AxisOP[1].AxisMotionPara.ReverseMotion_Velocity
            OnMouseClick: write the text variable via VisuDialogs.NumpadExtended
        Textfield (460,247 73x30), "%.3f", text variable: MAIN.AxisOP[3].AxisMotionPara.ReverseMotion_Velocity
            OnMouseClick: write the text variable via VisuDialogs.Numpad
        Textfield (555,247 73x30), "%.3f", text variable: MAIN.AxisOP[4].AxisMotionPara.ReverseMotion_Velocity
            OnMouseClick: write the text variable via VisuDialogs.Numpad
        Textfield (654,247 73x30), "%.3f", text variable: MAIN.AxisOP[5].AxisMotionPara.ReverseMotion_Velocity
            OnMouseClick: write the text variable via VisuDialogs.Numpad
        Textfield (365,211 73x30), "%.3f", text variable: MAIN.AxisOP[2].AxisMotionPara.TargetPosition2
            OnMouseClick: write the text variable via VisuDialogs.Numpad
        Textfield (270,211 73x30), "%.3f", text variable: MAIN.AxisOP[1].AxisMotionPara.TargetPosition2
            OnMouseClick: write the text variable via VisuDialogs.Numpad
        Textfield (460,211 73x30), "%.3f", text variable: MAIN.AxisOP[3].AxisMotionPara.TargetPosition2
            OnMouseClick: write the text variable via VisuDialogs.Numpad
        Textfield (555,211 73x30), "%.3f", text variable: MAIN.AxisOP[4].AxisMotionPara.TargetPosition2
            OnMouseClick: write the text variable via VisuDialogs.Numpad
        Textfield (654,211 73x30), "%.3f", text variable: MAIN.AxisOP[5].AxisMotionPara.TargetPosition2
            OnMouseClick: write the text variable via VisuDialogs.Numpad
        Label (54,212 113x30), "TargetPosition2/°:"
        Lamp1 (570,120 38x40), variable: MAIN.AxisOP[4].move_reverse_lamp, style: Lamp-Lamp1-Yellow
        Lamp1 (672,121 38x40), variable: MAIN.AxisOP[5].move_reverse_lamp, style: Lamp-Lamp1-Yellow
    Button (856,830 65x50), "home"
        tap MAIN.home
END_VISUALIZATION

(* stored: Version 1.1.0.1, ProductVersion 3.1.4024.12
   Visu StatJoint_6Axis: Id {493dabaa-a47e-493a-8617-dec037aa8fc6} *)
